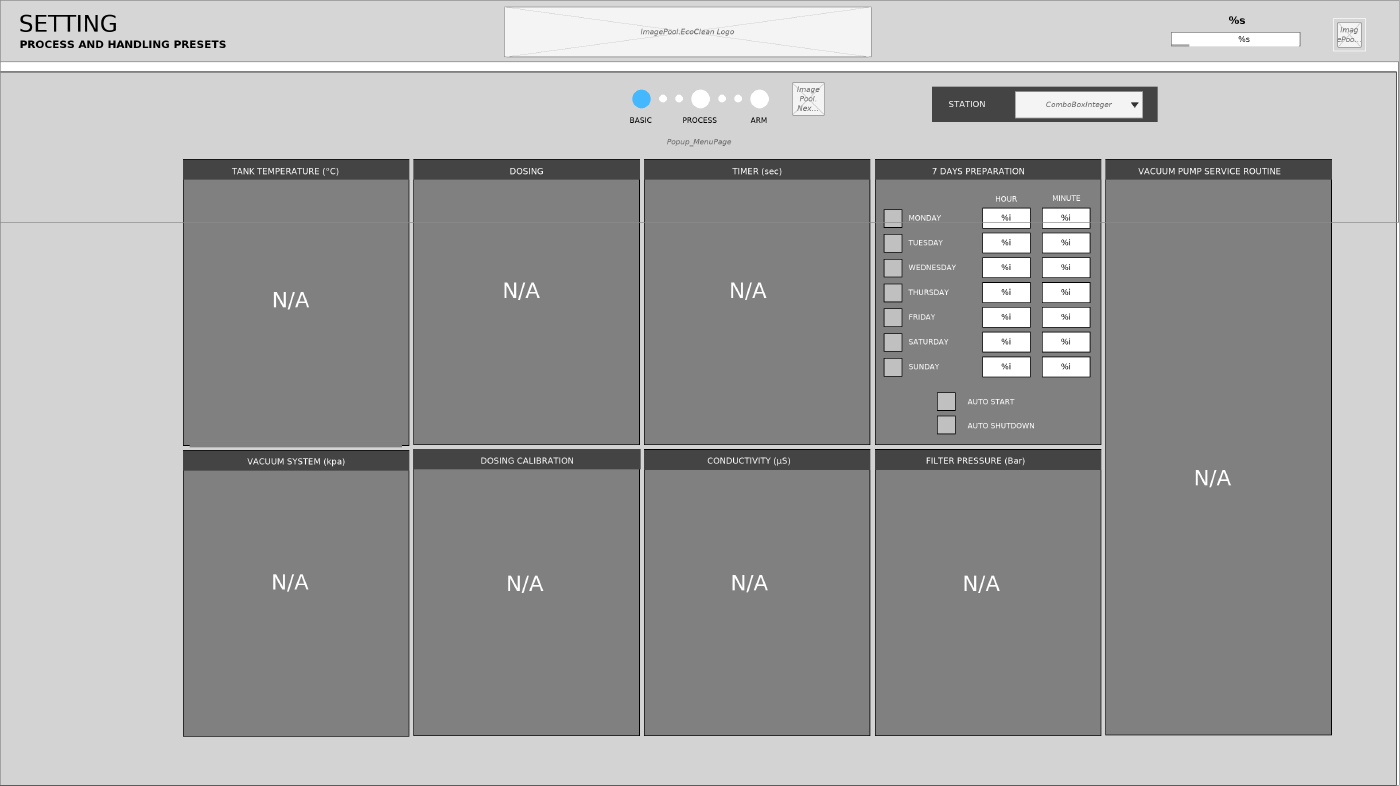
VISUALIZATION Setting_Page  // 1920x1078
    Rectangle (0,98 1915x980)
    Rectangle (0,63 1920x26)
        p3528305787: HMI_Ctrl.ANIMATION3
    Rectangle (0,0 1919x85)
    Label (23,6 267x53), "SETTING"
    Label (24,49 320x24), "PROCESS AND HANDLING PRESETS"
    Group (1828,25 45x45)
        OnMouseClick: toggle HMI_Ctrl.MenuButton
        RoundedRectangle (0,0 45x45), colour toggle: HMI_Ctrl.MenuButton
        Image (6,5 33x35), image: ImagePool.Menu Button
    Ellipse (867,123 25x25)
    Ellipse (948,123 25x25)
    Ellipse (904,130 10x10)
    Ellipse (926,130 10x10)
    Ellipse (985,130 10x10)
    Ellipse (1007,130 10x10)
    Ellipse (1029,123 25x25)
    Label (847,153 64x24), "BASIC"
    Label (928,153 64x24), "PROCESS"
    Label (1009,153 64x24), "ARM"
    Image (1086,113 45x45), image: ImagePool.Next Button
        OnMouseClick: change screen: SettingProcess_Page
    Rectangle (883,218 310x392)
    Rectangle (883,219 310x27)
    Label (967,223 143x24), "TIMER (sec)"
    Label (897,262 153x24), "TEMP NOT READY ALARM", invisible if: iSettingStnNoBuffer=0 OR iSettingStnNoBuffer=8 OR iSettingStnNoBuffer=5 OR iSettingStnNoBuffer=11
    Label (897,293 108x24), "DRIPPING TIME", invisible if: iSettingStnNoBuffer=0 OR iSettingStnNoBuffer=8 OR iSettingStnNoBuffer=11
    Label (897,324 196x24), "BAD BASKET TOLERANCE TIME", invisible if: iSettingStnNoBuffer=0 OR iSettingStnNoBuffer=8 OR iSettingStnNoBuffer=11
    Label (897,355 186x24), "INCOMING VALVE DELAY OFF", invisible if: iSettingStnNoBuffer=0 OR iSettingStnNoBuffer=9 OR iSettingStnNoBuffer=8 OR iSettingStnNoBuffer=6
    Rectangle (1081,265 119x17), "%i", text variable: ARiStnPreparationTempSv[iSettingStnNo], invisible if: iSettingStnNoBuffer=0 OR iSettingStnNoBuffer=8 OR iSettingStnNoBuffer=5 OR iSettingStnNoBuffer=11, input disabled if: bMainOnOff
        OnMouseDown: write the text variable via VisuDialogs.Numpad, min iStnPreparationTempMINsvHMIDisplay, max iStnPreparationTempMAXSVHMIDisplay
    Rectangle (1081,295 119x17), "%i", text variable: ARiStnDippingTimeSV[iSettingStnNo], invisible if: iSettingStnNoBuffer=0 OR iSettingStnNoBuffer=8 OR iSettingStnNoBuffer=11, input disabled if: bMainOnOff
        OnMouseDown: write the text variable via VisuDialogs.Numpad, min 0, max 100
    Rectangle (1081,325 119x17), "%i", text variable: ARiStnToleranceTimeSV[iSettingStnNo], invisible if: iSettingStnNoBuffer=0 OR iSettingStnNoBuffer=8 OR iSettingStnNoBuffer=11, input disabled if: bMainOnOff
        OnMouseDown: write the text variable via VisuDialogs.Numpad, min 0, max 999
    Rectangle (1081,355 119x17), "%i", text variable: ARiStnTopUpDelayOffTimeSV[iSettingStnNo], invisible if: iSettingStnNoBuffer=0 OR iSettingStnNoBuffer=9 OR iSettingStnNoBuffer=8 OR iSettingStnNoBuffer=6, input disabled if: bMainOnOff
        OnMouseDown: write the text variable via VisuDialogs.Numpad, min 0, max 20
    Label (897,385 186x24), "UNLOADING BUZZER", invisible if: iSettingStnNoBuffer<>8
    Rectangle (1081,387 119x17), "%i", text variable: diUnloadingSingleBasketReachedTimer, invisible if: iSettingStnNoBuffer<>8, input disabled if: bMainOnOff
        OnMouseDown: write the text variable via VisuDialogs.Numpad, min 10, max 999
    RoundedRectangle (1278,119 309x48)
    Label (1298,131 79x24), "STATION"
    ComboBoxInteger (1392,125 175x37), variable: iSettingStnNoBuffer, text list: 'TextList_SettingPage'
    Rectangle (1200,218 310x392)
    Rectangle (1200,219 310x27)
    Label (1275,223 161x24), "7 DAYS PREPARATION"
    Label (1243,287 93x24), "MONDAY"
    RoundedRectangle (1347,285 66x28), "%i", text variable: Day1H[OnOffStatus], invisible if: NOT.Day1En[OnOffStatus], input disabled if: bMainOnOff
        OnMouseDown: write the text variable via VisuDialogs.Keypad, min 0, max 23
    Label (1349,261 62x24), "HOUR"
    Label (1429,260 67x24), "MINUTE"
    Label (1243,321 93x24), "TUESDAY"
    Label (1243,355 93x24), "WEDNESDAY"
    Label (1243,389 93x24), "THURSDAY"
    Label (1243,423 93x24), "FRIDAY"
    Label (1243,457 93x24), "SATURDAY"
    Label (1243,491 93x24), "SUNDAY"
    Label (1324,539 93x24), "AUTO START"
    Label (1324,572 120x24), "AUTO SHUTDOWN"
    RoundedRectangle (1347,319 66x28), "%i", text variable: Day2H[OnOffStatus], invisible if: NOT.Day2En[OnOffStatus], input disabled if: bMainOnOff
        OnMouseDown: write the text variable via VisuDialogs.Keypad, min 0, max 23
    RoundedRectangle (1347,353 66x28), "%i", text variable: Day3H[OnOffStatus], invisible if: NOT.Day3En[OnOffStatus], input disabled if: bMainOnOff
        OnMouseDown: write the text variable via VisuDialogs.Keypad, min 0, max 23
    RoundedRectangle (1347,387 66x28), "%i", text variable: Day4H[OnOffStatus], invisible if: NOT.Day4En[OnOffStatus], input disabled if: bMainOnOff
        OnMouseDown: write the text variable via VisuDialogs.Keypad, min 0, max 23
    RoundedRectangle (1347,421 66x28), "%i", text variable: Day5H[OnOffStatus], invisible if: NOT.Day5En[OnOffStatus], input disabled if: bMainOnOff
        OnMouseDown: write the text variable via VisuDialogs.Keypad, min 0, max 23
    RoundedRectangle (1347,455 66x28), "%i", text variable: Day6H[OnOffStatus], invisible if: NOT.Day6En[OnOffStatus], input disabled if: bMainOnOff
        OnMouseDown: write the text variable via VisuDialogs.Keypad, min 0, max 23
    RoundedRectangle (1347,489 66x28), "%i", text variable: Day7H[OnOffStatus], invisible if: NOT.Day7En[OnOffStatus], input disabled if: bMainOnOff
        OnMouseDown: write the text variable via VisuDialogs.Keypad, min 0, max 23
    RoundedRectangle (1429,285 66x28), "%i", text variable: Day1M[OnOffStatus], invisible if: NOT.Day1En[OnOffStatus], input disabled if: bMainOnOff
        OnMouseDown: write the text variable via VisuDialogs.Keypad, min 0, max 59
    RoundedRectangle (1429,319 66x28), "%i", text variable: Day2M[OnOffStatus], invisible if: NOT.Day2En[OnOffStatus], input disabled if: bMainOnOff
        OnMouseDown: write the text variable via VisuDialogs.Keypad, min 0, max 59
    RoundedRectangle (1429,353 66x28), "%i", text variable: Day3M[OnOffStatus], invisible if: NOT.Day3En[OnOffStatus], input disabled if: bMainOnOff
        OnMouseDown: write the text variable via VisuDialogs.Keypad, min 0, max 59
    RoundedRectangle (1429,387 66x28), "%i", text variable: Day4M[OnOffStatus], invisible if: NOT.Day4En[OnOffStatus], input disabled if: bMainOnOff
        OnMouseDown: write the text variable via VisuDialogs.Keypad, min 0, max 59
    RoundedRectangle (1429,421 66x28), "%i", text variable: Day5M[OnOffStatus], invisible if: NOT.Day5En[OnOffStatus], input disabled if: bMainOnOff
        OnMouseDown: write the text variable via VisuDialogs.Keypad, min 0, max 59
    RoundedRectangle (1429,455 66x28), "%i", text variable: Day6M[OnOffStatus], invisible if: NOT.Day6En[OnOffStatus], input disabled if: bMainOnOff
        OnMouseDown: write the text variable via VisuDialogs.Keypad, min 0, max 59
    RoundedRectangle (1429,489 66x28), "%i", text variable: Day7M[OnOffStatus], invisible if: NOT.Day7En[OnOffStatus], input disabled if: bMainOnOff
        OnMouseDown: write the text variable via VisuDialogs.Keypad, min 0, max 59
    Rectangle (1212,287 25x25), colour toggle: Day1En[OnOffStatus], input disabled if: bMainOnOff
        toggle Day1En[OnOffStatus]
    Rectangle (1212,321 25x25), colour toggle: Day2En[OnOffStatus], input disabled if: bMainOnOff
        toggle Day2En[OnOffStatus]
    Rectangle (1212,355 25x25), colour toggle: Day3En[OnOffStatus], input disabled if: bMainOnOff
        toggle Day3En[OnOffStatus]
    Rectangle (1212,389 25x25), colour toggle: Day4En[OnOffStatus], input disabled if: bMainOnOff
        toggle Day4En[OnOffStatus]
    Rectangle (1212,423 25x25), colour toggle: Day5En[OnOffStatus], input disabled if: bMainOnOff
        toggle Day5En[OnOffStatus]
    Rectangle (1212,457 25x25), colour toggle: Day6En[OnOffStatus], input disabled if: bMainOnOff
        toggle Day6En[OnOffStatus]
    Rectangle (1212,491 25x25), colour toggle: Day7En[OnOffStatus], input disabled if: bMainOnOff
        toggle Day7En[OnOffStatus]
    Rectangle (1285,538 25x25), colour toggle: OnOffStatus=1
        OnMouseDown: execute { OnOffStatus:=1; }
    Rectangle (1285,570 25x25), colour toggle: OnOffStatus=2
        OnMouseDown: execute { OnOffStatus:=2; }
    Rectangle (567,616 310x393)
    Label (582,667 167x28), "CALIBRATE FEED (pulse)"
    Rectangle (779,665 82x28), "%i", text variable: ARDSProminentDosingHMI[iSettingStnNo].In_iCalibrateFeed_Pulse, input disabled if: bMainOnOff
        OnMouseDown: write the text variable via VisuDialogs.Numpad, min 10, max 999
    Label (586,707 159x28), "CALIBRATE RESULT (ml)"
    Rectangle (779,705 82x28), "%i", text variable: ARDSProminentDosingHMI[iSettingStnNo].In_iCalibrateTotalVolumeResult_ml, input disabled if: bMainOnOff
        OnMouseDown: write the text variable via VisuDialogs.Numpad, min 1, max 9999
    Label (586,747 159x28), "CALIBRATE START"
    Rectangle (757,748 110x30), "START", colour toggle: ARDSProminentDosingHMI[iSettingStnNo].In_bCalibratePB, input disabled if: bMainOnOff
        toggle ARDSProminentDosingHMI[iSettingStnNo].In_bCalibratePB
    Rectangle (773,886 74x30), "RESET", colour toggle: ARDSProminentDosingHMI[iSettingStnNo].In_bResetRemainedDosingVolumePB, input disabled if: bMainOnOff
        tap ARDSProminentDosingHMI[HMI_Ctrl.StationInfoPageNo].In_bResetRemainedDosingVolumePB
    Label (588,888 129x28), "RESET REMAINING DOSING VOLUME (ml)"
    Label (586,797 159x28), "CALIBRATE IN PROGRESS"
    Label (586,837 159x28), "CALIBRATE DONE"
    Ellipse (807,795 25x25), colour toggle: ARDSProminentDosingHMI[iSettingStnNo].Out_bCalibrateInProgress
    Ellipse (807,835 25x25), colour toggle: ARDSProminentDosingHMI[iSettingStnNo].Out_bCalibrateDone
    Group (581,653 291x349), invisible if: iSettingStnNoBuffer<>0 AND iSettingStnNoBuffer<>5 AND iSettingStnNoBuffer<>6 AND iSettingStnNoBuffer<>7 AND iSettingStnNoBuffer<>8 AND iSettingStnNoBuffer<>9
        Rectangle (0,0 291x349)
        Label (110,122 81x51), "N/A"
    Rectangle (568,616 310x27)
    Label (635,618 176x28), "DOSING CALIBRATION"
    Rectangle (567,218 310x392)
    Rectangle (567,219 310x27)
    Label (651,221 143x28), "DOSING"
    Label (581,262 129x28), "DOSE PER PULSE (ml)"
    Label (581,299 159x28), "VOLUME PER BASKET (ml)"
    Label (581,336 224x28), "NUMBER OF BASKET BETWEEN DOSING"
    Label (584,373 118x28), "REMAINING DOSING VOLUME (ml)"
    Label (581,460 91x28), "FIRST FILL (ml)"
    Rectangle (768,261 82x28), "%0.02f", text variable: ARDSProminentDosingHMI[iSettingStnNo].In_rVolumePerPulse_ml, input disabled if: bMainOnOff
    Rectangle (768,301 82x28), "%i", text variable: ARDSProminentDosingHMI[iSettingStnNo].In_iVolumePerBasket_ml, input disabled if: bMainOnOff
        OnMouseDown: write the text variable via VisuDialogs.Numpad, min 1, max 9999
    Rectangle (768,331 82x28), "%i", text variable: ARDSProminentDosingHMI[iSettingStnNo].In_iNoOfBasketBetweenAutoDosing, input disabled if: bMainOnOff
        OnMouseDown: write the text variable via VisuDialogs.Numpad, min 1, max 999
    Rectangle (770,369 82x28), "%0.01f", text variable: ARDSProminentDosingHMI[iSettingStnNo].Out_rRemainedDosingVolume_ml
    Rectangle (768,458 82x28), "%i", text variable: ARDSProminentDosingHMI[iSettingStnNo].in_iFirstFillDosing_ml, input disabled if: bMainOnOff
        OnMouseDown: write the text variable via VisuDialogs.Numpad, min 1, max 32767
    Label (584,424 118x28), "TOTALIZER DOSING VOLUME"
    Rectangle (803,420 70x28), "%i", text variable: ARDSProminentDosingHMI[iSettingStnNo].Out_iDosingTotalizer_ml
    Label (581,501 129x28), "RESET REMAINING DOSING VOLUME (ml)"
    Rectangle (768,499 74x30), "RESET", colour toggle: ARDSProminentDosingHMI[iSettingStnNo].In_bResetRemainedDosingVolumePB, input disabled if: bMainOnOff
        tap ARDSProminentDosingHMI[iSettingStnNo].In_bResetRemainedDosingVolumePB
    Label (580,551 152x28), "RESET REMAINING DOSING TOTALIZER (ml)"
    Rectangle (767,549 74x30), "RESET", colour toggle: ARDSProminentDosingHMI[iSettingStnNo].In_bResetDosingTotalizerPB, input disabled if: bMainOnOff
        tap ARDSProminentDosingHMI[iSettingStnNo].In_bResetDosingTotalizerPB
    Rectangle (883,616 310x393)
    Rectangle (883,617 310x27)
    Label (967,620 143x24), "CONDUCTIVITY (μS)"
    Label (896,661 108x24), "ACTUAL VALUE"
    Rectangle (1018,662 169x17), "%0.01f", text variable: ARrStnConductivityPV[iSettingStnNo]
    Rectangle (1018,693 169x17), "%0.01f", text variable: ARrStnLowConductivitySv[iSettingStnNo], input disabled if: bMainOnOff
        OnMouseDown: write the text variable via VisuDialogs.Numpad, min 0, max 999
    Rectangle (1018,723 169x17), "%0.01f", text variable: ARrStnHighConductivitySv[iSettingStnNo], input disabled if: bMainOnOff
        OnMouseDown: write the text variable via VisuDialogs.Numpad, min 0, max 99999
    Rectangle (895,692 119x17), "LOW ALARM", text variable: sDisplayConductivity[1]
    Rectangle (895,722 119x17), "HIGH ALARM", text variable: sDisplayConductivity[2]
    Group (889,652 291x349), invisible if: iSettingStnNoBuffer=5
        Rectangle (0,0 291x349)
        Label (110,122 81x51), "N/A"
    Rectangle (1200,616 310x393)
    Rectangle (1200,617 310x27)
    Label (1267,620 177x24), "FILTER PRESSURE (Bar)"
    Label (1212,661 108x24), "ACTUAL VALUE"
    Rectangle (1334,662 169x17), "%0.01f", text variable: ARrStnFilterPressurePV[iSettingStnNo]
    Rectangle (1334,693 169x17), "%0.01f", text variable: ARrStnLowFilterPressureSv[iSettingStnNo], input disabled if: bMainOnOff
        OnMouseDown: write the text variable via VisuDialogs.Numpad, min 0, max 999
    Rectangle (1334,723 169x17), "%0.01f", text variable: ARrStnHighFilterPressureSv[iSettingStnNo], input disabled if: bMainOnOff
        OnMouseDown: write the text variable via VisuDialogs.Numpad, min 0, max 999
    Label (1212,691 108x24), "LOW ALARM"
    Label (1212,720 108x24), "HIGH ALARM"
    Group (1207,653 291x349), invisible if: iSettingStnNoBuffer<> 6 AND iSettingStnNoBuffer<> 7 AND iSettingStnNoBuffer<> 8 AND iSettingStnNoBuffer<> 9
        Rectangle (0,0 291x349)
        Label (110,122 81x51), "N/A"
    Rectangle (251,218 310x393)
    Rectangle (251,219 310x27)
    Label (315,223 183x24), "TANK TEMPERATURE (°C)"
    Label (265,262 109x24), "SET VALUE", invisible if: iSettingStnNoBuffer=5
    Label (265,293 108x24), "ACTUAL VALUE"
    Label (265,324 116x24), "HIGH TEMP ALARM", invisible if: iSettingStnNoBuffer=5
    Label (265,355 133x24), "1ST LIMIT ALARM (+/-)", invisible if: iSettingStnNoBuffer=5
    Label (265,385 82x24), "HYSTERESIS", invisible if: iSettingStnNoBuffer=5
    Label (265,416 82x24), "READY (+/-)", invisible if: iSettingStnNoBuffer=5
    Rectangle (387,266 169x17), "%0.01f", text variable: ARrStnTempSV[iSettingStnNo], invisible if: iSettingStnNoBuffer=5, input disabled if: bMainOnOff
        OnMouseDown: write the text variable via VisuDialogs.Numpad, min rStnTempMINsvHMIDisplay, max rStnTempMAXsvHMIDisplay
    Rectangle (387,297 169x17), "%0.01f", text variable: ARrStnTempPV[iSettingStnNo]
    Rectangle (387,328 169x17), "%0.01f", text variable: ARrStnTempHALsv[iSettingStnNo], invisible if: iSettingStnNoBuffer=5, input disabled if: bMainOnOff
        OnMouseDown: write the text variable via VisuDialogs.Numpad, min rStnTempHALMINsvHMIDisplay, max rStnTempHALMAXsvHMIDisplay
    Rectangle (387,359 169x17), "%0.01f", text variable: ARrStnTemp1stLimitSv[iSettingStnNo], invisible if: iSettingStnNoBuffer=5, input disabled if: bMainOnOff
        OnMouseDown: write the text variable via VisuDialogs.Numpad, min rStnTemp1stLimitMINsvHMIDisplay, max rStnTemp1stLimitMAXsvHMIDisplay
    Rectangle (387,389 169x17), "%0.01f", text variable: ARrStnTempHYSsv[iSettingStnNo], invisible if: iSettingStnNoBuffer=5, input disabled if: bMainOnOff
        OnMouseDown: write the text variable via VisuDialogs.Numpad, min rStnTempHYSMINsvHMIDisplay, max rStnTempHYSMAXsvHMIDisplay
    Rectangle (387,420 169x17), "%0.01f", text variable: ARrStnTempRDYsv[iSettingStnNo], invisible if: iSettingStnNoBuffer=5, input disabled if: bMainOnOff
        OnMouseDown: write the text variable via VisuDialogs.Numpad, min rStnTempRDYMINsvHMIDisplay, max rStnTempRDYMAXsvHMIDisplay
    Group (260,264 291x332), invisible if: iSettingStnNoBuffer<>7 AND iSettingStnNoBuffer<>8 AND iSettingStnNoBuffer<>9
        Rectangle (0,0 291x349)
        Label (110,122 81x51), "N/A"
    Rectangle (251,617 310x393)
    Rectangle (251,618 310x27)
    Label (298,621 217x24), "VACUUM SYSTEM (kpa)"
    Image (691,9 504x69), image: ImagePool.EcoClean Logo
    Group (1606,17 179x46)
        Button (0,27 177x19), image: VisuSymbols.Symbols.AddUser
        Rectangle (25,28 150x18), "%s", text variable: fbHmiTF1800_UserlevelManagement.dsHmiUserStatus_Active.sLoginName
        Rectangle (2,0 177x22), "%s", text variable: DSLocalSystemTimeML.sCurrentDT24Hr_General
    Rectangle (720,420 82x28), "%i", text variable: ARDSProminentDosingHMI[iSettingStnNo].Out_iDosingTotalizer_Litre
    Label (756,398 24x28), "L"
    Label (821,398 24x28), "ml"
    Group (576,251 291x346), invisible if: iSettingStnNoBuffer<>0 AND iSettingStnNoBuffer<>5 AND iSettingStnNoBuffer<>6 AND iSettingStnNoBuffer<>7 AND iSettingStnNoBuffer<>8 AND iSettingStnNoBuffer<>9
        Rectangle (0,0 291x349)
        Label (110,122 81x51), "N/A"
    Group (887,251 291x346), invisible if: iSettingStnNoBuffer<>0 AND iSettingStnNoBuffer<>7 AND iSettingStnNoBuffer<>9
        Rectangle (0,0 291x349)
        Label (110,122 81x51), "N/A"
    Label (267,661 108x24), "VACUUM LEVEL"
    Rectangle (389,662 169x17), "%0.01f", text variable: ARrStnVacuumPV[iSettingStnNo]
    Rectangle (389,693 169x17), "%0.01f", text variable: ARrStnHighVacuumLevelSV[iSettingStnNo], input disabled if: bMainOnOff
        OnMouseDown: write the text variable via VisuDialogs.Numpad, min -120, max 10
    Rectangle (389,723 169x17), "%0.01f", text variable: ARrStnLowVacuumLevelSV[iSettingStnNo], input disabled if: bMainOnOff
        OnMouseDown: write the text variable via VisuDialogs.Numpad, min -120, max 10
    Rectangle (266,692 119x17), "HIGH VACUUM LEVEL", text variable: sDisplayConductivity[1]
    Rectangle (266,722 119x17), "LOW VACUUM LEVEL", text variable: sDisplayConductivity[2]
    Group (259,651 291x349), invisible if: iSettingStnNoBuffer= 6
        Rectangle (0,0 291x349)
        Label (110,122 81x51), "N/A"
    Rectangle (1516,218 310x790)
    Rectangle (1516,219 310x27)
    Label (1558,223 233x24), "VACUUM PUMP SERVICE ROUTINE"
    Label (1530,263 177x24), "VACUUM PUMP SERVICE HOUR"
    Rectangle (1741,327 58x17), "%i", text variable: ARdiVacPump2ndLimitTimerSV[iSettingStnNo], input disabled if: iCurrentUserGroupID<6 OR bMainOnOff
        OnMouseDown: write the text variable via VisuDialogs.Numpad, min 0, max 999
    Label (1530,321 92x24), "2nd LIMIT TIMER"
    Label (1530,383 159x24), "VACUUM PUMP TIMER"
    Rectangle (1745,379 57x24), "RESET", colour toggle: ARDSProminentDosingHMI[iSettingStnNo].In_bResetRemainedDosingVolumePB, input disabled if: iCurrentUserGroupID<6 OR bMainOnOff
        tap ARbVacuumPumpTimerReset[iSettingStnNo]
    Label (1530,349 159x24), "VACUUM PUMP RUN TIMER"
    Rectangle (1731,353 78x17), "%s", text variable: ARsVacuumPumpRunningTime[iSettingStnNo]
    Label (1530,293 92x24), "1st LIMIT TIMER"
    Rectangle (1741,299 58x17), "%i", text variable: ARdiVacPump1stLimitTimerSV[iSettingStnNo], input disabled if: iCurrentUserGroupID<6 OR bMainOnOff
        OnMouseDown: write the text variable via VisuDialogs.Numpad, min 0, max 999
    Label (1530,433 248x24), "VACUUM PUMP ROUTINE SERVICE DAYS"
    Rectangle (1741,497 58x17), "%i", text variable: ARiAlarmDaysSV_Routine[iSettingStnNo], input disabled if: iCurrentUserGroupID<6 OR bMainOnOff
        OnMouseDown: write the text variable via VisuDialogs.Numpad, min 0, max 999
    Label (1530,491 92x24), "2nd LIMIT TIMER"
    Label (1530,553 159x24), "VACUUM PUMP TIMER"
    Rectangle (1745,549 57x24), "RESET", colour toggle: ARDSProminentDosingHMI[iSettingStnNo].In_bResetRemainedDosingVolumePB, input disabled if: iCurrentUserGroupID<6 OR bMainOnOff
        tap ARbDaysPvReset_Routine[6]
    Label (1530,519 159x24), "VACUUM PUMP RUN TIMER"
    Rectangle (1731,523 78x17), "%i", text variable: ARiRunDaysPV_Routine[iSettingStnNo]
    Label (1530,463 92x24), "1st LIMIT TIMER"
    Rectangle (1741,469 58x17), "%i", text variable: ARiWarningDaysSV_Routine[iSettingStnNo], input disabled if: iCurrentUserGroupID<6 OR bMainOnOff
        OnMouseDown: write the text variable via VisuDialogs.Numpad, min 0, max 999
    Label (1530,613 227x24), "VACUUM PUMP MAJOR SERVICE DAYS"
    Rectangle (1741,677 58x17), "%i", text variable: ARiAlarmDaysSV_Major[iSettingStnNo], input disabled if: iCurrentUserGroupID<6 OR bMainOnOff
        OnMouseDown: write the text variable via VisuDialogs.Numpad, min 0, max 999
    Label (1530,671 92x24), "2nd LIMIT TIMER"
    Label (1530,733 159x24), "VACUUM PUMP TIMER"
    Rectangle (1745,729 57x24), "RESET", colour toggle: ARDSProminentDosingHMI[iSettingStnNo].In_bResetRemainedDosingVolumePB, input disabled if: iCurrentUserGroupID<6 OR bMainOnOff
        tap ARbDaysPvReset_Major[6]
    Label (1530,699 159x24), "VACUUM PUMP RUN TIMER"
    Rectangle (1731,703 78x17), "%i", text variable: ARiRunDaysPV_Major[iSettingStnNo]
    Label (1530,643 92x24), "1st LIMIT TIMER"
    Rectangle (1741,649 58x17), "%i", text variable: ARiWarningDaysSV_Major[iSettingStnNo], input disabled if: iCurrentUserGroupID<6 OR bMainOnOff
        OnMouseDown: write the text variable via VisuDialogs.Numpad, min 0, max 999
    Group (1526,259 283x735), invisible if: iSettingStnNoBuffer=6
        Rectangle (0,0 283x735)
        Label (108,372 74x49), "N/A"
    Frame (0,84 1918x221), invisible if: HMI_Ctrl.CloseMenuButton
        shows Popup_MenuPage()
END_VISUALIZATION

(* stored: Version 1.1.0.1, ProductVersion 3.1.4024.12
   Visu Setting_Page: Id {7948bd3a-0176-428f-83f9-b20d16f8d64b} *)
